TYPE (* Funk_DI Struct *)
  (* Version 1.0, 2025-07-21, Franz Höpfinger, initial API and implementation and/or initial documentation *)
  PACKAGE Funk::io::DI;
  IMPORT eclipse4diac::core::TypeHash;
  Funk_DI_S : STRUCT
    Pin : SINT := 127;
  END_STRUCT;
END_TYPE
